FUNCTION_BLOCK PID_HMI (* Service Interface Function Block Type *)
  (* Standard: 61499-2 *)
  (* Version 0.0, 1/20/2026, Schneider Electric, template *)
  PACKAGE Hidryco.HidrycoLib;
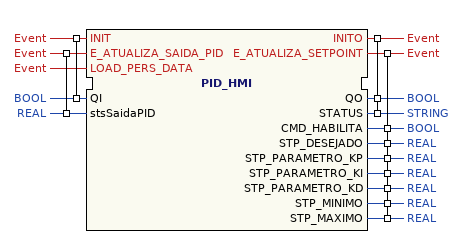
  EVENT_INPUT
    INIT WITH QI;
    E_ATUALIZA_SAIDA_PID WITH stsSaidaPID;
    LOAD_PERS_DATA;
  END_EVENT
  EVENT_OUTPUT
    INITO WITH QO, STATUS;
    E_ATUALIZA_SETPOINT WITH CMD_HABILITA, STP_DESEJADO, STP_PARAMETRO_KP, STP_PARAMETRO_KI, STP_PARAMETRO_KD, STP_MAXIMO, STP_MINIMO;
  END_EVENT
  VAR_INPUT
    QI : BOOL;
    stsSaidaPID : REAL;
  END_VAR
  VAR_OUTPUT
    QO : BOOL; (* Event Output Qualifier *)
    STATUS : STRING; (* Service Status *)
    CMD_HABILITA : BOOL;
    STP_DESEJADO : REAL;
    STP_PARAMETRO_KP : REAL;
    STP_PARAMETRO_KI : REAL;
    STP_PARAMETRO_KD : REAL;
    STP_MINIMO : REAL;
    STP_MAXIMO : REAL;
  END_VAR
  SERVICE /
    SEQUENCE 
    END_SEQUENCE
  END_SERVICE
END_FUNCTION_BLOCK
